(*

.. <legal notes>

legal notes
=================
| SPDX-FileCopyrightText: © 2025 Oleksandr Tiutyk <trofimich@gmail.com>
| SPDX-License-Identifier: LGPL-3.0-only
| For details check: LGPL-3.0-only_

.. _LGPL-3.0-only: https://www.gnu.org/licenses/lgpl-3.0.en.html

.. </legal notes>

*)

INTERFACE IComparer EXTENDS IObject

METHOD Compare : COMPARISION_RESULT
VAR_INPUT
	first : __SYSTEM.AnyType;
	second : __SYSTEM.AnyType;
END_VAR
END_METHOD

END_INTERFACE

(* stored: Version 1.1.0.1
   Itf IComparer: Id {610e5cb7-c530-4689-b27d-7bafa4915f53}
   Method Compare: Id {9e540de8-35be-4ff8-92e5-2183140bd76b} *)
